FUNCTION_BLOCK FB_AlarmEvent
VAR_INPUT
	bAlarmEvent		:BOOL;
	bButtAlarmReset	:BOOL;
END_VAR
VAR_IN_OUT
	fbAlarm		  :FB_TcAlarm;
END_VAR

IF bAlarmEvent THEN	
	fbAlarm.Raise(0);
END_IF
IF bButtAlarmReset THEN	
	fbAlarm.Clear(0, TRUE);
END_IF

END_FUNCTION_BLOCK

(* stored: Version 1.1.0.1, ProductVersion 3.1.4024.4
   POU FB_AlarmEvent: Id {e697f7dc-bc41-4499-8580-166f28536191}, SpecialFunc None *)
